KUKA KRL program: f_fraes_3.src, f_fraes_3.dat

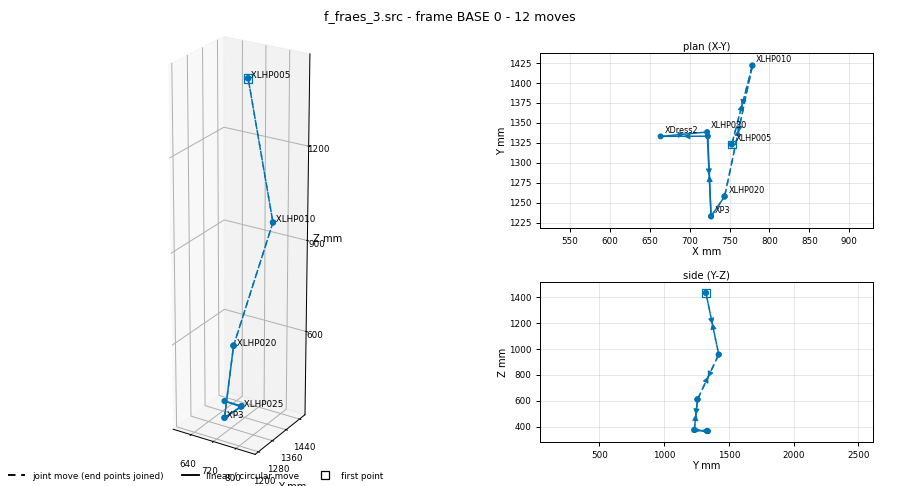
[picture p0: tool path of f_fraes_3.src in frame BASE 0, 12 of 12 moves have a stored position in this frame; points joined in program order, loops and branches not executed]
--- f_fraes_3.src ---
&ACCESS RVO7
&REL 6
&COMMENT Fresa C2
&PARAM DISKPATH = KRC:\R1\Program
&PARAM TEMPLATE = C:\KRC\Roboter\Template\vorgabe
&PARAM EDITMASK = *
DEF f_fraes_3( )
;FOLD INI
   ;FOLD BASISTECH INI
      GLOBAL INTERRUPT DECL 3 WHEN $STOPMESS==TRUE DO IR_STOPM ( )
      INTERRUPT ON 3
      BAS (#INITMOV,0 )
   ;ENDFOLD (BASISTECH INI)
   ;FOLD SPOTTECH INI
      USERSPOT(#INIT)
   ;ENDFOLD (SPOTTECH INI)
   ;FOLD GRIPPERTECH INI
      USER_GRP(0,DUMMY,DUMMY,GDEFAULT)
   ;ENDFOLD (GRIPPERTECH INI)
   ;FOLD USER INI
      ;Make your modifications here

   ;ENDFOLD (USER INI)
;ENDFOLD (INI)

; Estacao P13.060 - Robo R1
; Programa: Fresa C2
; Caracterização dos meios de produção:

chk_w3_wechs_ok ( )   ; CHECK FERRAMENTA: GUN C2

;FOLD PTP LHP005 Vel=100 % PDAT15 Tool[3]:GUN C2 Base[0];%{PE}%R 8.2.20,%MKUKATPBASIS,%CMOVE,%VPTP,%P 1:PTP, 2:LHP005, 3:, 5:100, 7:PDAT15
$BWDSTART=FALSE
PDAT_ACT=PPDAT15
FDAT_ACT=FLHP005
BAS(#PTP_PARAMS,100)
PTP XLHP005
;ENDFOLD
;FOLD PTP LHP010 CONT Vel=100 % PDAT16 Tool[3]:GUN C2 Base[0];%{PE}%R 8.2.20,%MKUKATPBASIS,%CMOVE,%VPTP,%P 1:PTP, 2:LHP010, 3:C_DIS, 5:100, 7:PDAT16
$BWDSTART=FALSE
PDAT_ACT=PPDAT16
FDAT_ACT=FLHP010
BAS(#PTP_PARAMS,100)
PTP XLHP010 C_DIS
;ENDFOLD
;FOLD PTP LHP020 CONT Vel=100 % PDAT17 Tool[3]:GUN C2 Base[0];%{PE}%R 8.2.20,%MKUKATPBASIS,%CMOVE,%VPTP,%P 1:PTP, 2:LHP020, 3:C_DIS, 5:100, 7:PDAT17
$BWDSTART=FALSE
PDAT_ACT=PPDAT17
FDAT_ACT=FLHP020
BAS(#PTP_PARAMS,100)
PTP XLHP020 C_DIS
;ENDFOLD
;FOLD LIN P3 Vel=0.4 m/s CPDAT7 Tool[3]:GUN C2 Base[0];%{PE}%R 8.2.20,%MKUKATPBASIS,%CMOVE,%VLIN,%P 1:LIN, 2:P3, 3:, 5:0.4, 7:CPDAT7
$BWDSTART=FALSE
LDAT_ACT=LCPDAT7
FDAT_ACT=FP3
BAS(#CP_PARAMS,0.4)
LIN XP3
;ENDFOLD
;FOLD LIN LHP025 Vel=0.5 m/s CPDAT8 Tool[3]:GUN C2 Base[0];%{PE}%R 8.2.20,%MKUKATPBASIS,%CMOVE,%VLIN,%P 1:LIN, 2:LHP025, 3:, 5:0.5, 7:CPDAT8
$BWDSTART=FALSE
LDAT_ACT=LCPDAT8
FDAT_ACT=FLHP025
BAS(#CP_PARAMS,0.5)
LIN XLHP025
;ENDFOLD

;FOLD ; PONTO DE FRESAGEM;%{PE}%R 4.1.16,%MKUKATPBASIS,%CCOMMENT,%VNORMAL,%P 2:PONTO DE FRESAGEM
;ENDFOLD
;FOLD TIP.LIN_ Dress2, Spot Gun 2 , RETR open , Tool[3], Base[0], EXT.TCP=FALSE;%{PE}%MKUKATPUSER
FDAT_ACT=FDress2
BAS(#FRAMES)
LIN  XDress2
S_ACT.GUN=2
S_ACT.RETR=#opn
S_READY=FALSE
USERSPOT (#DRESS,S_ACT )
WAIT FOR  S_READY
;ENDFOLD

;FOLD LIN LHP030 Vel=0.4 m/s CPDAT3 Tool[3]:GUN C2 Base[0];%{PE}%R 8.2.20,%MKUKATPBASIS,%CMOVE,%VLIN,%P 1:LIN, 2:LHP030, 3:, 5:0.4, 7:CPDAT3
$BWDSTART=FALSE
LDAT_ACT=LCPDAT3
FDAT_ACT=FLHP030
BAS(#CP_PARAMS,0.4)
LIN XLHP030
;ENDFOLD
;FOLD LIN LHP035 Vel=0.5 m/s CPDAT4 Tool[3]:GUN C2 Base[0];%{PE}%R 8.2.20,%MKUKATPBASIS,%CMOVE,%VLIN,%P 1:LIN, 2:LHP035, 3:, 5:0.5, 7:CPDAT4
$BWDSTART=FALSE
LDAT_ACT=LCPDAT4
FDAT_ACT=FLHP035
BAS(#CP_PARAMS,0.5)
LIN XLHP035
;ENDFOLD
;FOLD PTP P5 CONT Vel=100 % PDAT18 Tool[3]:GUN C2 Base[0];%{PE}%R 8.2.20,%MKUKATPBASIS,%CMOVE,%VPTP,%P 1:PTP, 2:P5, 3:C_DIS, 5:100, 7:PDAT18
$BWDSTART=FALSE
PDAT_ACT=PPDAT18
FDAT_ACT=FP5
BAS(#PTP_PARAMS,100)
PTP XP5 C_DIS
;ENDFOLD

;FOLD PTP pSOLDA PDAT19 SPOT Gun=2 RETR OPN PgNo1=252 ACTIVE=1 Tool[3]:GUN C2 Base[0];%{PE}%R 8.2.2,%MKUKATPSPOT,%CSPOT,%VPTP,%P 1:PTP, 2:pSOLDA, 3:, 5:100, 7:PDAT19, 10:2, 12:#FIRST, 14:#OPN, 16:252, 18:1, 20:0, 22:0, 24:1, 25:NORMAL
$BWDSTART=FALSE
PDAT_ACT=PPDAT19
FDAT_ACT=FpSOLDA
BAS(#PTP_PARAMS,PPDAT19.VEL)
S_ACT.GUN=2
S_ACT.PAIR=SDEFAULT.PAIR
S_ACT.RETR=#OPN
S_ACT.CLO_TM=1
S_ACT.PGNO1=252
S_ACT.PGNO2=SDEFAULT.PGNO2
S_ACT.PRESS1=SDEFAULT.PRESS1
S_ACT.PRESS2=SDEFAULT.PRESS2
S_READY=FALSE
PTP XpSOLDA
USERSPOT(#SPOT, S_ACT)
WAIT FOR S_READY
;ENDFOLD

;FOLD PTP P4 CONT Vel=100 % PDAT6 Tool[3]:GUN C2 Base[0];%{PE}%R 8.2.20,%MKUKATPBASIS,%CMOVE,%VPTP,%P 1:PTP, 2:P4, 3:C_DIS, 5:100, 7:PDAT6
$BWDSTART=FALSE
PDAT_ACT=PPDAT6
FDAT_ACT=FP4
BAS(#PTP_PARAMS,100)
PTP XP4 C_DIS
;ENDFOLD
;FOLD PTP P6 Vel=100 % PDAT12 Tool[3]:GUN C2 Base[0];%{PE}%R 8.2.20,%MKUKATPBASIS,%CMOVE,%VPTP,%P 1:PTP, 2:P6, 3:, 5:100, 7:PDAT12
$BWDSTART=FALSE
PDAT_ACT=PPDAT12
FDAT_ACT=FP6
BAS(#PTP_PARAMS,100)
PTP XP6
;ENDFOLD

END

--- f_fraes_3.dat ---
&ACCESS RVO7
&REL 6
&COMMENT Fresa C2
&PARAM DISKPATH = KRC:\R1\Program
&PARAM TEMPLATE = C:\KRC\Roboter\Template\vorgabe
&PARAM EDITMASK = *
DEFDAT  f_fraes_3
;FOLD EXTERNAL DECLARATIONS;%{PE}%MKUKATPBASIS,%CEXT,%VCOMMON,%P
;FOLD GRIPPERTECH EXT
EXT  H50 (INT  :IN,INT  :IN,INT  :IN,GRP_TYP  :IN )
;ENDFOLD (GRIPPERTECH EXT)
;FOLD SPOTTECH EXT
EXT  USERSPOT (S_COMMAND  :IN,SPOT_TYPE  :IN )
;ENDFOLD (SPOTTECH EXT)
;FOLD BASISTECH EXT;%{PE}%MKUKATPBASIS,%CEXT,%VEXT,%P
EXT  BAS (BAS_COMMAND  :IN,REAL  :IN )
DECL INT SUCCESS
;ENDFOLD (BASISTECH EXT)
;FOLD USER EXT;%{E}%MKUKATPUSER,%CEXT,%VEXT,%P
;Make your modifications here

;ENDFOLD (USER EXT)
;ENDFOLD (EXTERNAL DECLARATIONS)

DECL E6POS XLHP010={X 778.625122,Y 1421.90503,Z 957.051025,A 94.8773117,B -7.357162,C -88.1516266,S 18,T 11,E1 0.0,E2 0.0,E3 0.0,E4 0.0,E5 0.0,E6 0.0}
DECL FDAT FLHP010={TOOL_NO 3,BASE_NO 0,IPO_FRAME #BASE,TQ_STATE FALSE}
DECL PDAT PPDAT1={VEL 100.0,ACC 100.0,APO_DIST 20.0,APO_MODE #CDIS}
DECL E6POS XLHP015={X 711.816284,Y 1199.59705,Z 384.370392,A 89.4471207,B 0.234582499,C -88.6843338,S 18,T 11,E1 0.0,E2 0.0,E3 0.0,E4 0.0,E5 0.0,E6 0.0}
DECL FDAT FLHP015={TOOL_NO 3,BASE_NO 0,IPO_FRAME #BASE,TQ_STATE FALSE}
DECL PDAT PPDAT2={VEL 100.0,ACC 100.0,APO_DIST 10.0,APO_MODE #CDIS}
DECL E6POS XLHP020={X 743.804871,Y 1257.95105,Z 610.852722,A 91.868103,B -3.18870711,C -87.7671738,S 18,T 11,E1 0.0,E2 0.0,E3 0.0,E4 0.0,E5 0.0,E6 0.0}
DECL FDAT FLHP020={TOOL_NO 3,BASE_NO 0,IPO_FRAME #BASE,TQ_STATE FALSE}
DECL PDAT PPDAT3={VEL 100.0,ACC 100.0,APO_DIST 5.0,APO_MODE #CDIS}
DECL E6POS XLHP025={X 722.834778,Y 1333.46106,Z 365.59259,A 90.9306335,B -3.44928288,C -88.4928207,S 18,T 11,E1 0.0,E2 0.0,E3 0.0,E4 0.0,E5 0.0,E6 0.0}
DECL FDAT FLHP025={TOOL_NO 3,BASE_NO 0,IPO_FRAME #BASE,TQ_STATE FALSE}
DECL LDAT LCPDAT1={VEL 2.0,ACC 100.0,APO_DIST 2.0,APO_FAC 50.0}
DECL FDAT FDress1={TOOL_NO 1,BASE_NO 0,IPO_FRAME #BASE}
DECL E6POS XDress1={X 100.2397,Y 1698.11304,Z 299.565399,A -134.933899,B 0.464014888,C -2.46981001,S 18,T 11,E1 0.0,E2 0.0,E3 0.0,E4 0.0,E5 0.0,E6 0.0}
DECL E6POS XPFRESA={X 100.2397,Y 1698.11304,Z 299.565399,A -134.933899,B 0.464014888,C -2.46981001,S 18,T 11,E1 0.0,E2 0.0,E3 0.0,E4 0.0,E5 0.0,E6 0.0}
DECL FDAT Fpfresa={TOOL_NO 1,BASE_NO 0,IPO_FRAME #BASE}
DECL LDAT LCPDAT2={VEL 2.0,ACC 100.0,APO_DIST 100.0,APO_FAC 50.0}
DECL E6POS XLHP030={X 721.936218,Y 1338.63696,Z 365.588287,A 90.9307098,B -3.44858503,C -88.4926224,S 22,T 19,E1 0.0,E2 0.0,E3 0.0,E4 0.0,E5 0.0,E6 0.0}
DECL FDAT FLHP030={TOOL_NO 3,BASE_NO 0,IPO_FRAME #BASE,TQ_STATE FALSE}
DECL LDAT LCPDAT3={VEL 2.0,ACC 100.0,APO_DIST 2.0,APO_FAC 50.0}
DECL E6POS XLHP035={X 726.905518,Y 1233.07202,Z 374.9534,A 91.8778,B -3.21575999,C -87.7657013,S 22,T 19,E1 0.0,E2 0.0,E3 0.0,E4 0.0,E5 0.0,E6 0.0}
DECL FDAT FLHP035={TOOL_NO 3,BASE_NO 0,IPO_FRAME #BASE,TQ_STATE FALSE}
DECL LDAT LCPDAT4={VEL 2.0,ACC 100.0,APO_DIST 10.0,APO_FAC 50.0}
DECL E6POS XLHP040={X 388.047913,Y 1486.42798,Z 838.35553,A 150.914307,B -0.181115806,C -18.4495907,S 18,T 3,E1 0.0,E2 0.0,E3 0.0,E4 0.0,E5 0.0,E6 0.0}
DECL FDAT FLHP040={TOOL_NO 1,BASE_NO 0,IPO_FRAME #BASE}
DECL PDAT PPDAT4={VEL 100.0,ACC 100.0,APO_DIST 15.0}
DECL E6POS XLHP045={X 388.052307,Y 1486.41003,Z 838.34668,A 150.907806,B -0.182964295,C -18.4479904,S 2,T 3,E1 0.0,E2 0.0,E3 0.0,E4 0.0,E5 0.0,E6 0.0}
DECL FDAT FLHP045={TOOL_NO 1,BASE_NO 0,IPO_FRAME #BASE}
DECL PDAT PPDAT5={VEL 100.0,ACC 100.0,APO_DIST 30.0}
DECL SPOT_SUGG_T LAST_SPOT={GUN[] "1                       ",RETR_CMD[] "#OPN                    ",CHOISE[] "#FIRST                  ",CLO_TM[] "1                       ",PGNO1[] "1                       ",PRESS1[] "0                       ",PGNO2[] "1                       ",PRESS2[] "0                       ",SPOT_PARAMS[] "NORMAL                  "}
DECL E6POS XPSOLDA={X 743.805481,Y 1257.99805,Z 610.852722,A 91.8718491,B -3.1881659,C -87.7667999,S 18,T 11,E1 0.0,E2 0.0,E3 0.0,E4 0.0,E5 0.0,E6 0.0}
DECL FDAT FpSOLDA={TOOL_NO 3,BASE_NO 0,IPO_FRAME #BASE,TQ_STATE FALSE}
DECL PDAT PPDAT7={VEL 50.0,ACC 100.0,APO_DIST 100.0}
DECL E6POS XLHP050={X 1325.32605,Y 356.201508,Z 900.299927,A 89.0204163,B 0.02457688,C -13.11127,S 18,T 3,E1 0.0,E2 0.0,E3 0.0,E4 0.0,E5 0.0,E6 0.0}
DECL FDAT FLHP050={TOOL_NO 1,BASE_NO 0,IPO_FRAME #BASE}
DECL PDAT PPDAT8={VEL 100.0,ACC 80.0,APO_DIST 10.0}
DECL PDAT PPDAT9={VEL 100.0,ACC 100.0,APO_DIST 10.0}
DECL E6POS XLHP005={X 752.775513,Y 1323.07703,Z 1432.68896,A 80.5145035,B -52.7116699,C -87.2903366,S 18,T 3,E1 0.0,E2 0.0,E3 0.0,E4 0.0,E5 0.0,E6 0.0}
DECL FDAT FLHP005={TOOL_NO 3,BASE_NO 0,IPO_FRAME #BASE,TQ_STATE FALSE}
DECL FDAT FDress2={TOOL_NO 3,BASE_NO 0,IPO_FRAME #BASE}
DECL E6POS XDress2={X 663.717224,Y 1333.17395,Z 368.721985,A 90.9740295,B -3.32114196,C -88.1314392,S 18,T 11,E1 0.0,E2 0.0,E3 0.0,E4 0.0,E5 0.0,E6 0.0}
DECL BASIS_SUGG_T LAST_BASIS={POINT1[] "PS01010001              ",POINT2[] "PS01010001              ",CP_PARAMS[] "CPDAT0                  ",PTP_PARAMS[] "PDAT0                   ",CONT[] "                        ",CP_VEL[] "2.0                     ",PTP_VEL[] " 100                    ",SPL_NAME[] "S0                      "}
DECL E6POS XP1={X 382.214813,Y 1646.07104,Z 258.947113,A 178.9245,B -0.858626127,C -0.883606017,S 18,T 11,E1 0.0,E2 0.0,E3 0.0,E4 0.0,E5 0.0,E6 0.0}
DECL FDAT FP1={TOOL_NO 1,BASE_NO 0,IPO_FRAME #BASE,POINT2[] " ",TQ_STATE FALSE}
DECL LDAT LCPDAT5={VEL 2.0,ACC 100.0,APO_DIST 100.0,APO_FAC 50.0,AXIS_VEL 100.0,AXIS_ACC 100.0,ORI_TYP #VAR,CIRC_TYP #BASE,JERK_FAC 50.0,GEAR_JERK 50.0,EXAX_IGN 0}
DECL E6POS XP2={X 255.032104,Y 1646.46802,Z 239.541595,A 178.911499,B -0.883683383,C -0.972572982,S 18,T 11,E1 0.0,E2 0.0,E3 0.0,E4 0.0,E5 0.0,E6 0.0}
DECL FDAT FP2={TOOL_NO 1,BASE_NO 0,IPO_FRAME #BASE,POINT2[] " ",TQ_STATE FALSE}
DECL LDAT LCPDAT6={VEL 2.0,ACC 100.0,APO_DIST 100.0,APO_FAC 50.0,AXIS_VEL 100.0,AXIS_ACC 100.0,ORI_TYP #VAR,CIRC_TYP #BASE,JERK_FAC 50.0,GEAR_JERK 50.0,EXAX_IGN 0}
DECL E6POS XP3={X 726.905518,Y 1233.07202,Z 374.9534,A 91.8778,B -3.21575999,C -87.7657013,S 22,T 19,E1 0.0,E2 0.0,E3 0.0,E4 0.0,E5 0.0,E6 0.0}
DECL FDAT FP3={TOOL_NO 3,BASE_NO 0,IPO_FRAME #BASE,POINT2[] " ",TQ_STATE FALSE}
DECL LDAT LCPDAT7={VEL 2.0,ACC 100.0,APO_DIST 100.0,APO_FAC 50.0,AXIS_VEL 100.0,AXIS_ACC 100.0,ORI_TYP #VAR,CIRC_TYP #BASE,JERK_FAC 50.0,GEAR_JERK 50.0,EXAX_IGN 0}
DECL E6POS XP4={X 778.625427,Y 1421.90698,Z 957.051514,A 94.8773117,B -7.35725498,C -88.1517563,S 18,T 11,E1 0.0,E2 0.0,E3 0.0,E4 0.0,E5 0.0,E6 0.0}
DECL FDAT FP4={TOOL_NO 3,BASE_NO 0,IPO_FRAME #BASE,POINT2[] " ",TQ_STATE FALSE}
DECL PDAT PPDAT6={VEL 100.0,ACC 100.0,APO_DIST 10.0,APO_MODE #CDIS,GEAR_JERK 50.0}
DECL E6POS XP5={X 743.804688,Y 1257.95496,Z 610.852722,A 91.8682404,B -3.18887496,C -87.7672119,S 18,T 11,E1 0.0,E2 0.0,E3 0.0,E4 0.0,E5 0.0,E6 0.0}
DECL FDAT FP5={TOOL_NO 3,BASE_NO 0,IPO_FRAME #BASE,POINT2[] " ",TQ_STATE FALSE}
DECL PDAT PPDAT10={VEL 100.0,ACC 100.0,APO_DIST 10.0,APO_MODE #CDIS,GEAR_JERK 50.0}
DECL PDAT PPDAT11={VEL 50.0,ACC 100.0,APO_DIST 100.0}
DECL E6POS XP6={X 752.775513,Y 1323.07703,Z 1432.68896,A 80.5145035,B -52.7116699,C -87.2903366,S 18,T 3,E1 0.0,E2 0.0,E3 0.0,E4 0.0,E5 0.0,E6 0.0}
DECL FDAT FP6={TOOL_NO 3,BASE_NO 0,IPO_FRAME #BASE,POINT2[] " ",TQ_STATE FALSE}
DECL PDAT PPDAT12={VEL 100.0,ACC 100.0,APO_DIST 100.0,APO_MODE #CDIS,GEAR_JERK 50.0}
DECL PDAT PPDAT13={VEL 50.0,ACC 100.0,APO_DIST 100.0}
DECL PDAT PPDAT14={VEL 100.0,ACC 100.0,APO_DIST 100.0,APO_MODE #CDIS,GEAR_JERK 50.0}
DECL LDAT LCPDAT8={VEL 2.0,ACC 100.0,APO_DIST 100.0,APO_FAC 50.0,AXIS_VEL 100.0,AXIS_ACC 100.0,ORI_TYP #VAR,CIRC_TYP #BASE,JERK_FAC 50.0,GEAR_JERK 50.0,EXAX_IGN 0}
DECL FDAT FDress3={TOOL_NO 3,BASE_NO 0,IPO_FRAME #BASE}
DECL E6POS XDress3={X 672.083984,Y 1337.797,Z 366.879913,A 90.9325333,B -3.44920802,C -88.4932632,S 22,T 19,E1 0.0,E2 0.0,E3 0.0,E4 0.0,E5 0.0,E6 0.0}
DECL LDAT LCPDAT9={VEL 2.0,ACC 100.0,APO_DIST 100.0,APO_FAC 50.0,AXIS_VEL 100.0,AXIS_ACC 100.0,ORI_TYP #VAR,CIRC_TYP #BASE,JERK_FAC 50.0,GEAR_JERK 50.0,EXAX_IGN 0}
DECL PDAT PPDAT15={VEL 100.0,ACC 100.0,APO_DIST 100.0,APO_MODE #CDIS,GEAR_JERK 50.0}
DECL LDAT LCPDAT10={VEL 2.0,ACC 100.0,APO_DIST 100.0,APO_FAC 50.0,AXIS_VEL 100.0,AXIS_ACC 100.0,ORI_TYP #VAR,CIRC_TYP #BASE,JERK_FAC 50.0,GEAR_JERK 50.0,EXAX_IGN 0}
DECL PDAT PPDAT16={VEL 100.0,ACC 100.0,APO_DIST 20.0,APO_MODE #CDIS,GEAR_JERK 50.0}
DECL LDAT LCPDAT11={VEL 2.0,ACC 100.0,APO_DIST 100.0,APO_FAC 50.0,AXIS_VEL 100.0,AXIS_ACC 100.0,ORI_TYP #VAR,CIRC_TYP #BASE,JERK_FAC 50.0,GEAR_JERK 50.0,EXAX_IGN 0}
DECL PDAT PPDAT17={VEL 100.0,ACC 100.0,APO_DIST 5.0,APO_MODE #CDIS,GEAR_JERK 50.0}
DECL LDAT LCPDAT12={VEL 2.0,ACC 100.0,APO_DIST 100.0,APO_FAC 50.0,AXIS_VEL 100.0,AXIS_ACC 100.0,ORI_TYP #VAR,CIRC_TYP #BASE,JERK_FAC 50.0,GEAR_JERK 50.0,EXAX_IGN 0}
DECL PDAT PPDAT18={VEL 100.0,ACC 100.0,APO_DIST 10.0,APO_MODE #CDIS,GEAR_JERK 50.0}
DECL LDAT LCPDAT13={VEL 2.0,ACC 100.0,APO_DIST 100.0,APO_FAC 50.0,AXIS_VEL 100.0,AXIS_ACC 100.0,ORI_TYP #VAR,CIRC_TYP #BASE,JERK_FAC 50.0,GEAR_JERK 50.0,EXAX_IGN 0}
DECL PDAT PPDAT19={VEL 50.0,ACC 100.0,APO_DIST 100.0,APO_MODE #CDIS,GEAR_JERK 50.0}
ENDDAT
